TYPE ST_AxisStruct :
STRUCT

///////Control from EPICS/NICOS/////////
///////Axis////////
    control     : ST_AxisControl;

///////Outputs/Status/////////
    status      : ST_AxisStatus;

///////Axis Parameters//////
    config      : ST_AxisConfig;

    description : ST_AxisDescription;

///////Axis Inputs///////
    inputs      : ST_AxisInputs;

///////Axis Ref///////
    Axis                :   AXIS_REF;       //The NC axis link to the hardware this is controlling

//////Gearing Parameters///////
    masterAxis          :   ST_GearAxis;                         //A reference to the axis that this is a slave of
    slaveAxisRatio      :   ARRAY [1..GVL_APP.nAXIS_NUM] OF LREAL; //The gearing between this axis as a master and any slaves. e.g. if this is a 1 to 1 master of axis 2 this will be [0, 1, 0 ...]

END_STRUCT
END_TYPE

(* stored: Version 1.1.0.1, ProductVersion 3.1.4024.0
   DUT ST_AxisStruct: Id {9732127f-85ab-48d1-a591-d13402fe3665} *)
